TYPE ST_DataSetEmulation :
(**************************************************************************************
 * 	Application		:	BoxControl Framework
 *	Revision		:	$Revision: 404529 $
 *	Revision date	:	$Date: 2018-04-23 08:21:38 +0200 (Mo., 23 Apr 2018) $
 *	Last changed by	:	$Author: b7bolm $
 *	URL				:	$URL: http://almscdc.swisslog.com/repo/SWPD/Development/BoxControlFramework/20_Release/trunk/01_Software/BCF/BCF/JumpStart/20_Product/11_Emu/10_Base/10_Lib/10_Conv/01_DUTs/ST_DataSetEmulation.TcDUT $
 *
 *	Purpose			:	TU Data - Data set - Emulation
 *
 * ------------------------------------------------------------------------------------
 *	Copyright Swisslog [IP AG], Switzerland. All rights reserved.
 * 
 * ------------------------------------------------------------------------------------
 *	
 * 	Revision History: 
 *
 * 	VERSION			DATE			INITIALS			DESCRIPTION
 *	0.1				01.01.2001		swl					Example
 *
 **************************************************************************************)
STRUCT
	DataPresent		: BOOL; // Data present
	LongSideLeading : BOOL; // TU runs long side leading
	NestedIndex		: DINT; // Index of nested data set
	ParentIndex		: DINT; // Index of parent in view of nested
 	Dimension		: ST_Dimension; // Dimensions
END_STRUCT
END_TYPE

(* stored: Version 1.1.0.1, ProductVersion 3.1.4022.12
   DUT ST_DataSetEmulation: Id {0d5679ec-e306-4aa0-b2ba-793d9c20f437} *)
